// TIA Portal V17 export
// export: Created 2023-07-20T16:54:09.9633399Z, ExportSetting WithDefaults, DisplayName Totally Integrated Automation Portal, DisplayVersion V17, DisplayName TIA Portal Openness, DisplayVersion V17, DisplayName TIA Portal Version Control Interface, DisplayVersion V17, DisplayName STEP 7 Professional, DisplayVersion V17, DisplayName STEP 7 Safety, DisplayVersion V17, DisplayName WinCC Professional, DisplayVersion V17
FUNCTION_BLOCK "Modbus RTU RW sequencer"   // FB1, LAD
{ S7_Optimized_Access := 'TRUE' }
VERSION : 0.1
// stored: AutoNumber false, IsIECCheckEnabled false, IsRetainMemResEnabled false, MemoryReserve 100, SetENOAutomatically false, UDAEnableTagReadback false
   VAR
      "Operation data number" { S7_SetPoint := 'True'} : "Deconcatenate UDInt into two UInt";
      "Operation type" { S7_SetPoint := 'True'} : "Deconcatenate UDInt into two UInt";
      Position { S7_SetPoint := 'True'} : "Deconcatenate UDInt into two UInt";
      Speed { S7_SetPoint := 'True'} : "Deconcatenate UDInt into two UInt";
      "Starting changing rate" { S7_SetPoint := 'True'} : "Deconcatenate UDInt into two UInt";
      "Stopping deceleration" { S7_SetPoint := 'True'} : "Deconcatenate UDInt into two UInt";
      "Operating current" { S7_SetPoint := 'True'} : "Deconcatenate UDInt into two UInt";
      "Operation trigger" { S7_SetPoint := 'True'} : "Deconcatenate UDInt into two UInt";
      "Forwarding destination" { S7_SetPoint := 'True'} : "Deconcatenate UDInt into two UInt";
      "Alarm reset" { S7_SetPoint := 'True'} : "Deconcatenate UDInt into two UInt";
      "Clear alarm history" { S7_SetPoint := 'True'} : "Deconcatenate UDInt into two UInt";
      "Clear comm history" { S7_SetPoint := 'True'} : "Deconcatenate UDInt into two UInt";
      "Clear monitor alarm history" { S7_SetPoint := 'True'} : "Deconcatenate UDInt into two UInt";
      "Clear comm history_1" { S7_SetPoint := 'True'} : "Deconcatenate UDInt into two UInt";
      "Monitor present alarm" { S7_SetPoint := 'True'} : "Concatenate two UInt into one UDInt";
      "Monitor alarm history 1" { S7_SetPoint := 'True'} : "Concatenate two UInt into one UDInt";
      "Monitor alarm history 2" { S7_SetPoint := 'True'} : "Concatenate two UInt into one UDInt";
      "Monitor alarm history 3" { S7_SetPoint := 'True'} : "Concatenate two UInt into one UDInt";
      "Monitor alarm history 4" { S7_SetPoint := 'True'} : "Concatenate two UInt into one UDInt";
      "Monitor alarm history 5" { S7_SetPoint := 'True'} : "Concatenate two UInt into one UDInt";
      "Monitor present communication error" { S7_SetPoint := 'True'} : "Concatenate two UInt into one UDInt";
      "Monitor communication error history 1" { S7_SetPoint := 'True'} : "Concatenate two UInt into one UDInt";
      "Monitor communication error history 2" { S7_SetPoint := 'True'} : "Concatenate two UInt into one UDInt";
      "Monitor communication error history 3" { S7_SetPoint := 'True'} : "Concatenate two UInt into one UDInt";
      "Monitor communication error history 4" { S7_SetPoint := 'True'} : "Concatenate two UInt into one UDInt";
      "Monitor communication error history 5" { S7_SetPoint := 'True'} : "Concatenate two UInt into one UDInt";
      "Monitor feedback position" { S7_SetPoint := 'True'} : "Concatenate two UInt into one UDInt";
      "Monitor feedback speed r/min" { S7_SetPoint := 'True'} : "Concatenate two UInt into one UDInt";
      "Monitor feedback speed Hz" { S7_SetPoint := 'True'} : "Concatenate two UInt into one UDInt";
      "Monitor direct I/O" { S7_SetPoint := 'True'} : "Concatenate two UInt into one UDInt";
      "Monitor torque" { S7_SetPoint := 'True'} : "Concatenate two UInt into one UDInt";
      "Monitor cumulative load" { S7_SetPoint := 'True'} : "Concatenate two UInt into one UDInt";
      "Monitor driver temperature" { S7_SetPoint := 'True'} : "Concatenate two UInt into one UDInt";
      "Monitor motor temperature" { S7_SetPoint := 'True'} : "Concatenate two UInt into one UDInt";
      "Monitor inverter voltage" { S7_SetPoint := 'True'} : "Concatenate two UInt into one UDInt";
      "Monitor power supply voltage" { S7_SetPoint := 'True'} : "Concatenate two UInt into one UDInt";
      "Monitor DIP SW" { S7_SetPoint := 'True'} : "Concatenate two UInt into one UDInt";
      "Monitor ROT SW0" { S7_SetPoint := 'True'} : "Concatenate two UInt into one UDInt";
      "Monitor ROT SW1" { S7_SetPoint := 'True'} : "Concatenate two UInt into one UDInt";
   END_VAR
   VAR_TEMP   // added for the SCL form of the ladder/FBD networks
      _w1 : Bool;
   END_VAR
BEGIN

REGION Network 1: Deconcatenate data for writing it into modbus holding registers
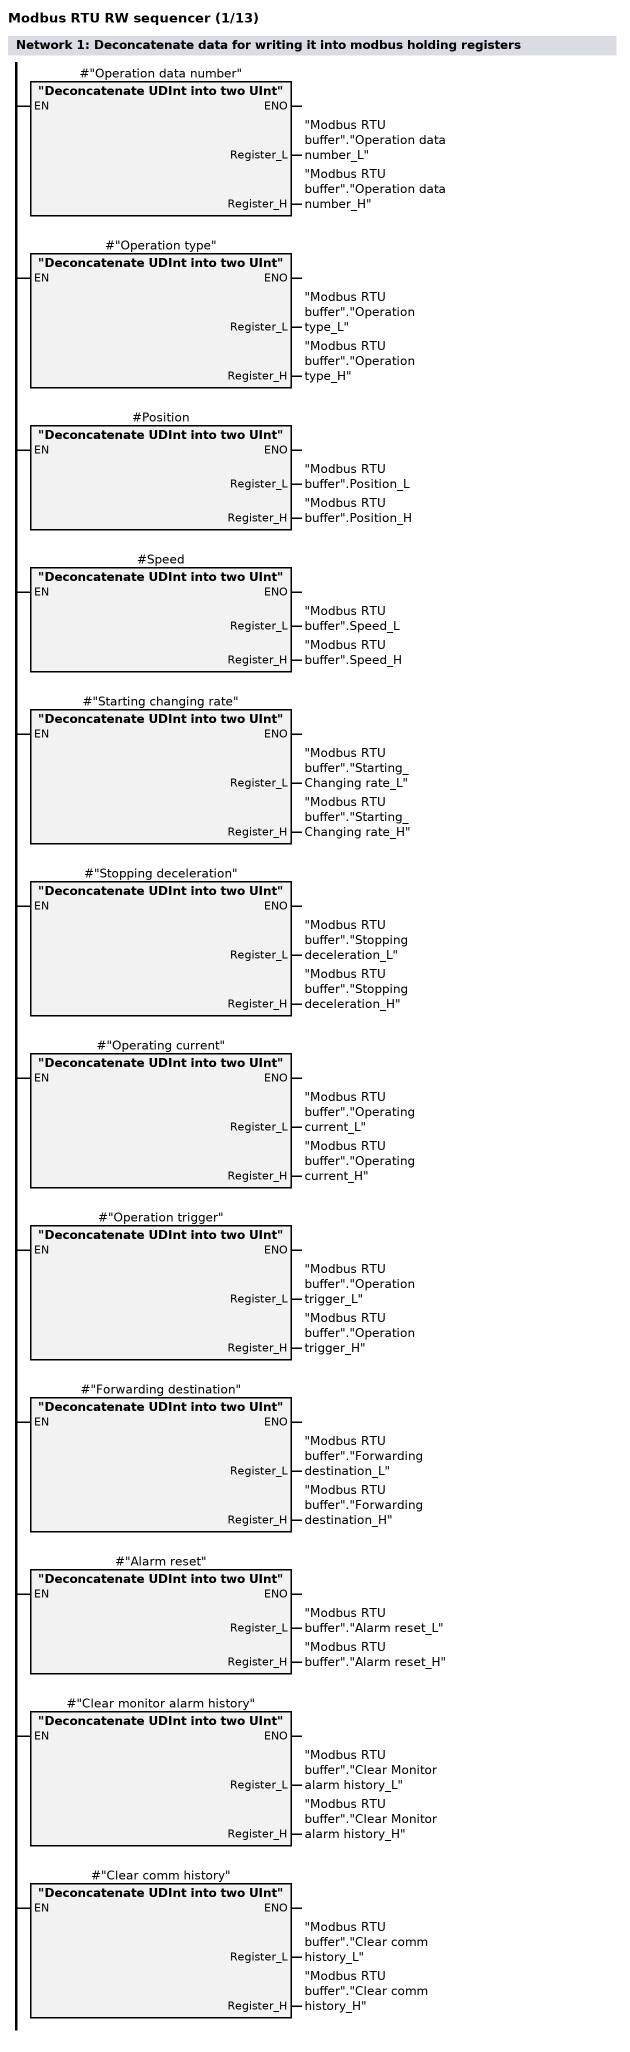
   RUNG wire#powerrail
      #"Operation data number"(Register_L => "Modbus RTU buffer"."Operation data number_L", Register_H => "Modbus RTU buffer"."Operation data number_H")
   END_RUNG
   RUNG wire#powerrail
      #"Operation type"(Register_L => "Modbus RTU buffer"."Operation type_L", Register_H => "Modbus RTU buffer"."Operation type_H")
   END_RUNG
   RUNG wire#powerrail
      #Position(Register_L => "Modbus RTU buffer".Position_L, Register_H => "Modbus RTU buffer".Position_H)
   END_RUNG
   RUNG wire#powerrail
      #Speed(Register_L => "Modbus RTU buffer".Speed_L, Register_H => "Modbus RTU buffer".Speed_H)
   END_RUNG
   RUNG wire#powerrail
      #"Starting changing rate"(Register_L => "Modbus RTU buffer"."Starting_Changing rate_L", Register_H => "Modbus RTU buffer"."Starting_Changing rate_H")
   END_RUNG
   RUNG wire#powerrail
      #"Stopping deceleration"(Register_L => "Modbus RTU buffer"."Stopping deceleration_L", Register_H => "Modbus RTU buffer"."Stopping deceleration_H")
   END_RUNG
   RUNG wire#powerrail
      #"Operating current"(Register_L => "Modbus RTU buffer"."Operating current_L", Register_H => "Modbus RTU buffer"."Operating current_H")
   END_RUNG
   RUNG wire#powerrail
      #"Operation trigger"(Register_L => "Modbus RTU buffer"."Operation trigger_L", Register_H => "Modbus RTU buffer"."Operation trigger_H")
   END_RUNG
   RUNG wire#powerrail
      #"Forwarding destination"(Register_L => "Modbus RTU buffer"."Forwarding destination_L", Register_H => "Modbus RTU buffer"."Forwarding destination_H")
   END_RUNG
   RUNG wire#powerrail
      #"Alarm reset"(Register_L => "Modbus RTU buffer"."Alarm reset_L", Register_H => "Modbus RTU buffer"."Alarm reset_H")
   END_RUNG
   RUNG wire#powerrail
      #"Clear monitor alarm history"(Register_L => "Modbus RTU buffer"."Clear Monitor alarm history_L", Register_H => "Modbus RTU buffer"."Clear Monitor alarm history_H")
   END_RUNG
   RUNG wire#powerrail
      #"Clear comm history"(Register_L => "Modbus RTU buffer"."Clear comm history_L", Register_H => "Modbus RTU buffer"."Clear comm history_H")
   END_RUNG
   // the same network as SCL:
   #"Operation data number"(Register_L => "Modbus RTU buffer"."Operation data number_L",   // "Deconcatenate UDInt into two UInt"
                           Register_H => "Modbus RTU buffer"."Operation data number_H");
   #"Operation type"(Register_L => "Modbus RTU buffer"."Operation type_L",   // "Deconcatenate UDInt into two UInt"
                     Register_H => "Modbus RTU buffer"."Operation type_H");
   #Position(Register_L => "Modbus RTU buffer".Position_L, Register_H => "Modbus RTU buffer".Position_H);   // "Deconcatenate UDInt into two UInt"
   #Speed(Register_L => "Modbus RTU buffer".Speed_L, Register_H => "Modbus RTU buffer".Speed_H);   // "Deconcatenate UDInt into two UInt"
   #"Starting changing rate"(Register_L => "Modbus RTU buffer"."Starting_Changing rate_L",   // "Deconcatenate UDInt into two UInt"
                           Register_H => "Modbus RTU buffer"."Starting_Changing rate_H");
   #"Stopping deceleration"(Register_L => "Modbus RTU buffer"."Stopping deceleration_L",   // "Deconcatenate UDInt into two UInt"
                           Register_H => "Modbus RTU buffer"."Stopping deceleration_H");
   #"Operating current"(Register_L => "Modbus RTU buffer"."Operating current_L",   // "Deconcatenate UDInt into two UInt"
                        Register_H => "Modbus RTU buffer"."Operating current_H");
   #"Operation trigger"(Register_L => "Modbus RTU buffer"."Operation trigger_L",   // "Deconcatenate UDInt into two UInt"
                        Register_H => "Modbus RTU buffer"."Operation trigger_H");
   #"Forwarding destination"(Register_L => "Modbus RTU buffer"."Forwarding destination_L",   // "Deconcatenate UDInt into two UInt"
                           Register_H => "Modbus RTU buffer"."Forwarding destination_H");
   #"Alarm reset"(Register_L => "Modbus RTU buffer"."Alarm reset_L",   // "Deconcatenate UDInt into two UInt"
                  Register_H => "Modbus RTU buffer"."Alarm reset_H");
   #"Clear monitor alarm history"(Register_L => "Modbus RTU buffer"."Clear Monitor alarm history_L",   // "Deconcatenate UDInt into two UInt"
                           Register_H => "Modbus RTU buffer"."Clear Monitor alarm history_H");
   #"Clear comm history"(Register_L => "Modbus RTU buffer"."Clear comm history_L",   // "Deconcatenate UDInt into two UInt"
                         Register_H => "Modbus RTU buffer"."Clear comm history_H");
END_REGION

REGION Network 2: Data writing/reading step 0: Write data from address 88 to address 105
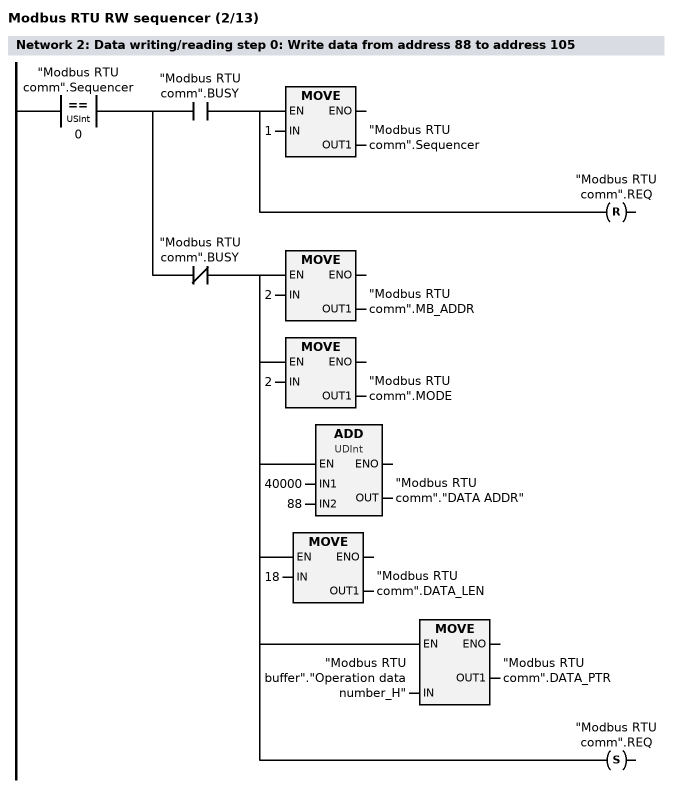
   RUNG wire#powerrail
      { S7_Templates := "SrcType := USInt" } EQ_Contact(in1 := "Modbus RTU comm".Sequencer, in2 := 0)
      wire#w1
      Contact( "Modbus RTU comm".BUSY )
      wire#w2
      Move(in := 1, out1 => "Modbus RTU comm".Sequencer)
   END_RUNG
   RUNG wire#w2
      R_Coil( "Modbus RTU comm".REQ )
   END_RUNG
   RUNG wire#w1
      I_Contact( "Modbus RTU comm".BUSY )
      wire#w3
      Move(in := 2, out1 => "Modbus RTU comm".MB_ADDR)
   END_RUNG
   RUNG wire#w3
      Move(in := 2, out1 => "Modbus RTU comm".MODE)
   END_RUNG
   RUNG wire#w3
      { S7_Templates := "SrcType := UDInt" } Add(in1 := 40000, in2 := 88, out => "Modbus RTU comm"."DATA ADDR")
   END_RUNG
   RUNG wire#w3
      Move(in := 18, out1 => "Modbus RTU comm".DATA_LEN)
   END_RUNG
   RUNG wire#w3
      Move(in := "Modbus RTU buffer"."Operation data number_H", out1 => "Modbus RTU comm".DATA_PTR)
   END_RUNG
   RUNG wire#w3
      S_Coil( "Modbus RTU comm".REQ )
   END_RUNG
   // the same network as SCL:
   #_w1 := "Modbus RTU comm".Sequencer = 0;
   IF #_w1 AND "Modbus RTU comm".BUSY THEN
       "Modbus RTU comm".Sequencer := 1;
       "Modbus RTU comm".REQ := FALSE;
   END_IF;
   IF #_w1 AND NOT "Modbus RTU comm".BUSY THEN
       "Modbus RTU comm".MB_ADDR := 2;
       "Modbus RTU comm".MODE := 2;
       "Modbus RTU comm"."DATA ADDR" := 40000 + 88;
       "Modbus RTU comm".DATA_LEN := 18;
       "Modbus RTU comm".DATA_PTR := "Modbus RTU buffer"."Operation data number_H";
       "Modbus RTU comm".REQ := TRUE;
   END_IF;
END_REGION

REGION Network 3: Data writing/reading step 1: Write data from address 384 to address 385
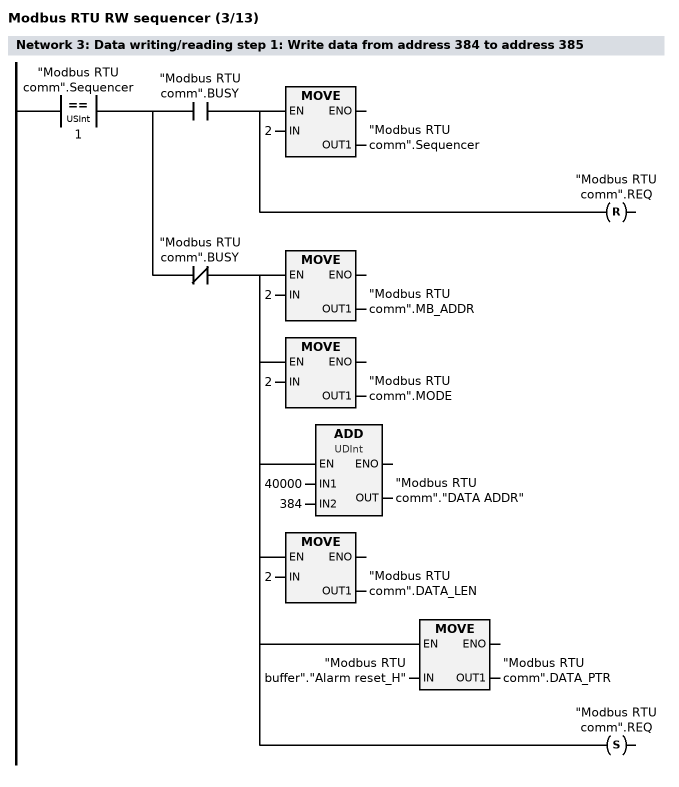
   RUNG wire#powerrail
      { S7_Templates := "SrcType := USInt" } EQ_Contact(in1 := "Modbus RTU comm".Sequencer, in2 := 1)
      wire#w1
      Contact( "Modbus RTU comm".BUSY )
      wire#w2
      Move(in := 2, out1 => "Modbus RTU comm".Sequencer)
   END_RUNG
   RUNG wire#w2
      R_Coil( "Modbus RTU comm".REQ )
   END_RUNG
   RUNG wire#w1
      I_Contact( "Modbus RTU comm".BUSY )
      wire#w3
      Move(in := 2, out1 => "Modbus RTU comm".MB_ADDR)
   END_RUNG
   RUNG wire#w3
      Move(in := 2, out1 => "Modbus RTU comm".MODE)
   END_RUNG
   RUNG wire#w3
      { S7_Templates := "SrcType := UDInt" } Add(in1 := 40000, in2 := 384, out => "Modbus RTU comm"."DATA ADDR")
   END_RUNG
   RUNG wire#w3
      Move(in := 2, out1 => "Modbus RTU comm".DATA_LEN)
   END_RUNG
   RUNG wire#w3
      Move(in := "Modbus RTU buffer"."Alarm reset_H", out1 => "Modbus RTU comm".DATA_PTR)
   END_RUNG
   RUNG wire#w3
      S_Coil( "Modbus RTU comm".REQ )
   END_RUNG
   // the same network as SCL:
   #_w1 := "Modbus RTU comm".Sequencer = 1;
   IF #_w1 AND "Modbus RTU comm".BUSY THEN
       "Modbus RTU comm".Sequencer := 2;
       "Modbus RTU comm".REQ := FALSE;
   END_IF;
   IF #_w1 AND NOT "Modbus RTU comm".BUSY THEN
       "Modbus RTU comm".MB_ADDR := 2;
       "Modbus RTU comm".MODE := 2;
       "Modbus RTU comm"."DATA ADDR" := 40000 + 384;
       "Modbus RTU comm".DATA_LEN := 2;
       "Modbus RTU comm".DATA_PTR := "Modbus RTU buffer"."Alarm reset_H";
       "Modbus RTU comm".REQ := TRUE;
   END_IF;
END_REGION

REGION Network 4: Data writing/reading step 2: Write data from address 388 to address 389
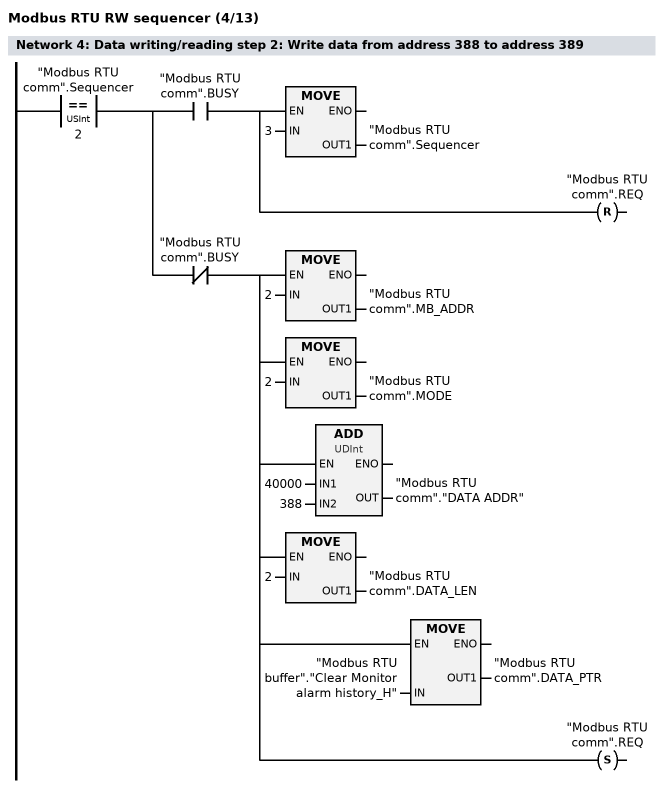
   RUNG wire#powerrail
      { S7_Templates := "SrcType := USInt" } EQ_Contact(in1 := "Modbus RTU comm".Sequencer, in2 := 2)
      wire#w1
      Contact( "Modbus RTU comm".BUSY )
      wire#w2
      Move(in := 3, out1 => "Modbus RTU comm".Sequencer)
   END_RUNG
   RUNG wire#w2
      R_Coil( "Modbus RTU comm".REQ )
   END_RUNG
   RUNG wire#w1
      I_Contact( "Modbus RTU comm".BUSY )
      wire#w3
      Move(in := 2, out1 => "Modbus RTU comm".MB_ADDR)
   END_RUNG
   RUNG wire#w3
      Move(in := 2, out1 => "Modbus RTU comm".MODE)
   END_RUNG
   RUNG wire#w3
      { S7_Templates := "SrcType := UDInt" } Add(in1 := 40000, in2 := 388, out => "Modbus RTU comm"."DATA ADDR")
   END_RUNG
   RUNG wire#w3
      Move(in := 2, out1 => "Modbus RTU comm".DATA_LEN)
   END_RUNG
   RUNG wire#w3
      Move(in := "Modbus RTU buffer"."Clear Monitor alarm history_H", out1 => "Modbus RTU comm".DATA_PTR)
   END_RUNG
   RUNG wire#w3
      S_Coil( "Modbus RTU comm".REQ )
   END_RUNG
   // the same network as SCL:
   #_w1 := "Modbus RTU comm".Sequencer = 2;
   IF #_w1 AND "Modbus RTU comm".BUSY THEN
       "Modbus RTU comm".Sequencer := 3;
       "Modbus RTU comm".REQ := FALSE;
   END_IF;
   IF #_w1 AND NOT "Modbus RTU comm".BUSY THEN
       "Modbus RTU comm".MB_ADDR := 2;
       "Modbus RTU comm".MODE := 2;
       "Modbus RTU comm"."DATA ADDR" := 40000 + 388;
       "Modbus RTU comm".DATA_LEN := 2;
       "Modbus RTU comm".DATA_PTR := "Modbus RTU buffer"."Clear Monitor alarm history_H";
       "Modbus RTU comm".REQ := TRUE;
   END_IF;
END_REGION

REGION Network 5: Data writing/reading step 3: Write data from address 392 to address 393
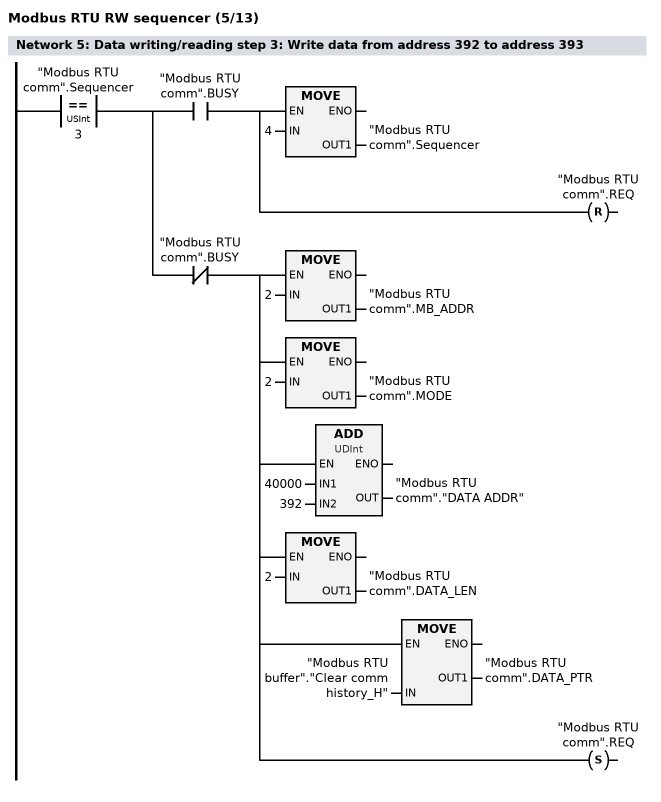
   RUNG wire#powerrail
      { S7_Templates := "SrcType := USInt" } EQ_Contact(in1 := "Modbus RTU comm".Sequencer, in2 := 3)
      wire#w1
      Contact( "Modbus RTU comm".BUSY )
      wire#w2
      Move(in := 4, out1 => "Modbus RTU comm".Sequencer)
   END_RUNG
   RUNG wire#w2
      R_Coil( "Modbus RTU comm".REQ )
   END_RUNG
   RUNG wire#w1
      I_Contact( "Modbus RTU comm".BUSY )
      wire#w3
      Move(in := 2, out1 => "Modbus RTU comm".MB_ADDR)
   END_RUNG
   RUNG wire#w3
      Move(in := 2, out1 => "Modbus RTU comm".MODE)
   END_RUNG
   RUNG wire#w3
      { S7_Templates := "SrcType := UDInt" } Add(in1 := 40000, in2 := 392, out => "Modbus RTU comm"."DATA ADDR")
   END_RUNG
   RUNG wire#w3
      Move(in := 2, out1 => "Modbus RTU comm".DATA_LEN)
   END_RUNG
   RUNG wire#w3
      Move(in := "Modbus RTU buffer"."Clear comm history_H", out1 => "Modbus RTU comm".DATA_PTR)
   END_RUNG
   RUNG wire#w3
      S_Coil( "Modbus RTU comm".REQ )
   END_RUNG
   // the same network as SCL:
   #_w1 := "Modbus RTU comm".Sequencer = 3;
   IF #_w1 AND "Modbus RTU comm".BUSY THEN
       "Modbus RTU comm".Sequencer := 4;
       "Modbus RTU comm".REQ := FALSE;
   END_IF;
   IF #_w1 AND NOT "Modbus RTU comm".BUSY THEN
       "Modbus RTU comm".MB_ADDR := 2;
       "Modbus RTU comm".MODE := 2;
       "Modbus RTU comm"."DATA ADDR" := 40000 + 392;
       "Modbus RTU comm".DATA_LEN := 2;
       "Modbus RTU comm".DATA_PTR := "Modbus RTU buffer"."Clear comm history_H";
       "Modbus RTU comm".REQ := TRUE;
   END_IF;
END_REGION

REGION Network 6: Data writing/reading step 4: Read data from address 128 to address 139
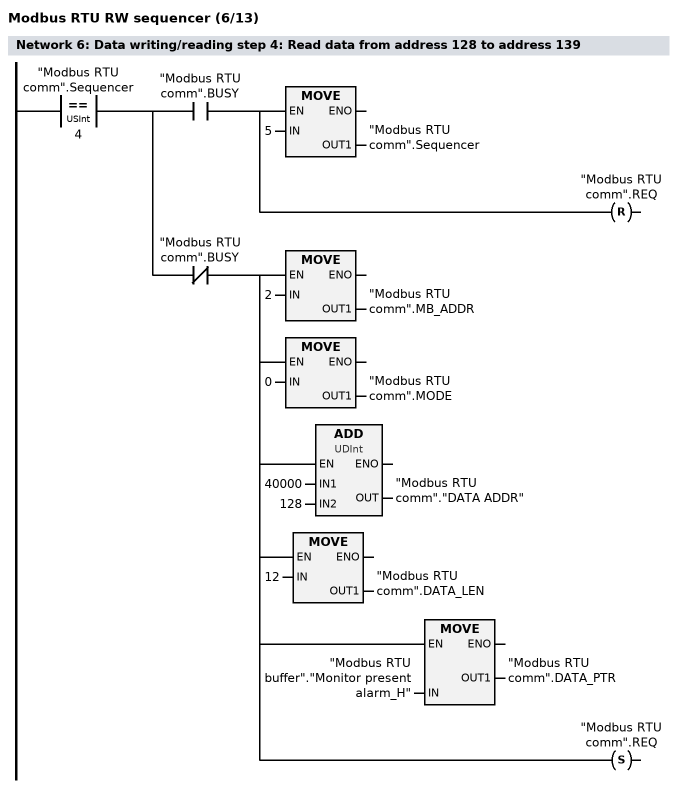
   RUNG wire#powerrail
      { S7_Templates := "SrcType := USInt" } EQ_Contact(in1 := "Modbus RTU comm".Sequencer, in2 := 4)
      wire#w1
      Contact( "Modbus RTU comm".BUSY )
      wire#w2
      Move(in := 5, out1 => "Modbus RTU comm".Sequencer)
   END_RUNG
   RUNG wire#w2
      R_Coil( "Modbus RTU comm".REQ )
   END_RUNG
   RUNG wire#w1
      I_Contact( "Modbus RTU comm".BUSY )
      wire#w3
      Move(in := 2, out1 => "Modbus RTU comm".MB_ADDR)
   END_RUNG
   RUNG wire#w3
      Move(in := 0, out1 => "Modbus RTU comm".MODE)
   END_RUNG
   RUNG wire#w3
      { S7_Templates := "SrcType := UDInt" } Add(in1 := 40000, in2 := 128, out => "Modbus RTU comm"."DATA ADDR")
   END_RUNG
   RUNG wire#w3
      Move(in := 12, out1 => "Modbus RTU comm".DATA_LEN)
   END_RUNG
   RUNG wire#w3
      Move(in := "Modbus RTU buffer"."Monitor present alarm_H", out1 => "Modbus RTU comm".DATA_PTR)
   END_RUNG
   RUNG wire#w3
      S_Coil( "Modbus RTU comm".REQ )
   END_RUNG
   // the same network as SCL:
   #_w1 := "Modbus RTU comm".Sequencer = 4;
   IF #_w1 AND "Modbus RTU comm".BUSY THEN
       "Modbus RTU comm".Sequencer := 5;
       "Modbus RTU comm".REQ := FALSE;
   END_IF;
   IF #_w1 AND NOT "Modbus RTU comm".BUSY THEN
       "Modbus RTU comm".MB_ADDR := 2;
       "Modbus RTU comm".MODE := 0;
       "Modbus RTU comm"."DATA ADDR" := 40000 + 128;
       "Modbus RTU comm".DATA_LEN := 12;
       "Modbus RTU comm".DATA_PTR := "Modbus RTU buffer"."Monitor present alarm_H";
       "Modbus RTU comm".REQ := TRUE;
   END_IF;
END_REGION

REGION Network 7: Data writing/reading step 5: Read data from address 172 to address 183
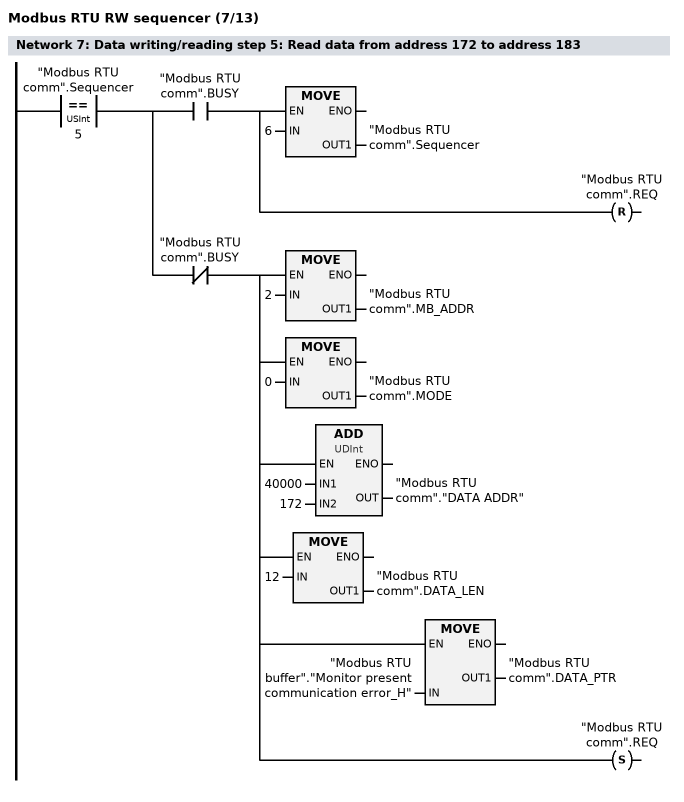
   RUNG wire#powerrail
      { S7_Templates := "SrcType := USInt" } EQ_Contact(in1 := "Modbus RTU comm".Sequencer, in2 := 5)
      wire#w1
      Contact( "Modbus RTU comm".BUSY )
      wire#w2
      Move(in := 6, out1 => "Modbus RTU comm".Sequencer)
   END_RUNG
   RUNG wire#w2
      R_Coil( "Modbus RTU comm".REQ )
   END_RUNG
   RUNG wire#w1
      I_Contact( "Modbus RTU comm".BUSY )
      wire#w3
      Move(in := 2, out1 => "Modbus RTU comm".MB_ADDR)
   END_RUNG
   RUNG wire#w3
      Move(in := 0, out1 => "Modbus RTU comm".MODE)
   END_RUNG
   RUNG wire#w3
      { S7_Templates := "SrcType := UDInt" } Add(in1 := 40000, in2 := 172, out => "Modbus RTU comm"."DATA ADDR")
   END_RUNG
   RUNG wire#w3
      Move(in := 12, out1 => "Modbus RTU comm".DATA_LEN)
   END_RUNG
   RUNG wire#w3
      Move(in := "Modbus RTU buffer"."Monitor present communication error_H", out1 => "Modbus RTU comm".DATA_PTR)
   END_RUNG
   RUNG wire#w3
      S_Coil( "Modbus RTU comm".REQ )
   END_RUNG
   // the same network as SCL:
   #_w1 := "Modbus RTU comm".Sequencer = 5;
   IF #_w1 AND "Modbus RTU comm".BUSY THEN
       "Modbus RTU comm".Sequencer := 6;
       "Modbus RTU comm".REQ := FALSE;
   END_IF;
   IF #_w1 AND NOT "Modbus RTU comm".BUSY THEN
       "Modbus RTU comm".MB_ADDR := 2;
       "Modbus RTU comm".MODE := 0;
       "Modbus RTU comm"."DATA ADDR" := 40000 + 172;
       "Modbus RTU comm".DATA_LEN := 12;
       "Modbus RTU comm".DATA_PTR := "Modbus RTU buffer"."Monitor present communication error_H";
       "Modbus RTU comm".REQ := TRUE;
   END_IF;
END_REGION

REGION Network 8: Data writing/reading step 6: Read data from address 204 to address 209
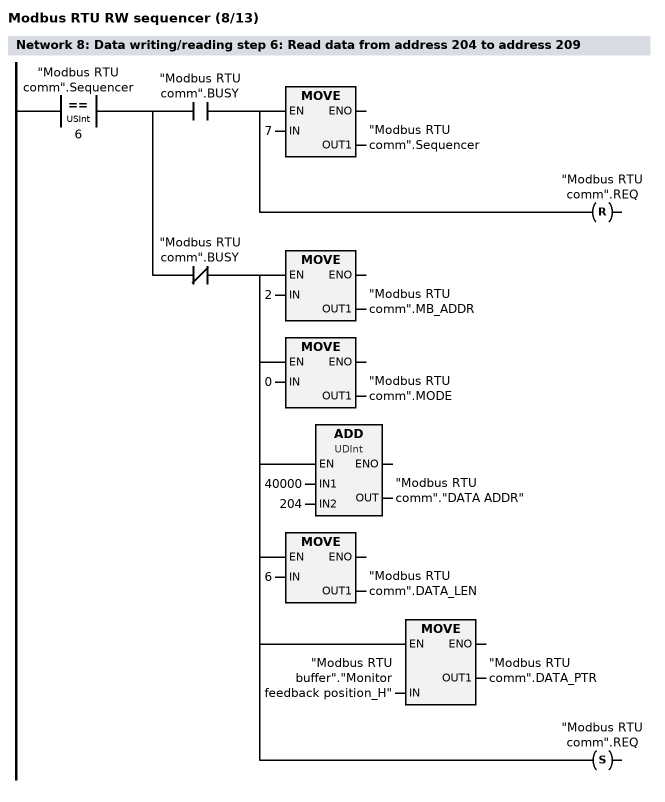
   RUNG wire#powerrail
      { S7_Templates := "SrcType := USInt" } EQ_Contact(in1 := "Modbus RTU comm".Sequencer, in2 := 6)
      wire#w1
      Contact( "Modbus RTU comm".BUSY )
      wire#w2
      Move(in := 7, out1 => "Modbus RTU comm".Sequencer)
   END_RUNG
   RUNG wire#w2
      R_Coil( "Modbus RTU comm".REQ )
   END_RUNG
   RUNG wire#w1
      I_Contact( "Modbus RTU comm".BUSY )
      wire#w3
      Move(in := 2, out1 => "Modbus RTU comm".MB_ADDR)
   END_RUNG
   RUNG wire#w3
      Move(in := 0, out1 => "Modbus RTU comm".MODE)
   END_RUNG
   RUNG wire#w3
      { S7_Templates := "SrcType := UDInt" } Add(in1 := 40000, in2 := 204, out => "Modbus RTU comm"."DATA ADDR")
   END_RUNG
   RUNG wire#w3
      Move(in := 6, out1 => "Modbus RTU comm".DATA_LEN)
   END_RUNG
   RUNG wire#w3
      Move(in := "Modbus RTU buffer"."Monitor feedback position_H", out1 => "Modbus RTU comm".DATA_PTR)
   END_RUNG
   RUNG wire#w3
      S_Coil( "Modbus RTU comm".REQ )
   END_RUNG
   // the same network as SCL:
   #_w1 := "Modbus RTU comm".Sequencer = 6;
   IF #_w1 AND "Modbus RTU comm".BUSY THEN
       "Modbus RTU comm".Sequencer := 7;
       "Modbus RTU comm".REQ := FALSE;
   END_IF;
   IF #_w1 AND NOT "Modbus RTU comm".BUSY THEN
       "Modbus RTU comm".MB_ADDR := 2;
       "Modbus RTU comm".MODE := 0;
       "Modbus RTU comm"."DATA ADDR" := 40000 + 204;
       "Modbus RTU comm".DATA_LEN := 6;
       "Modbus RTU comm".DATA_PTR := "Modbus RTU buffer"."Monitor feedback position_H";
       "Modbus RTU comm".REQ := TRUE;
   END_IF;
END_REGION

REGION Network 9: Data writing/reading step 7: Read data from address 212 to address 215
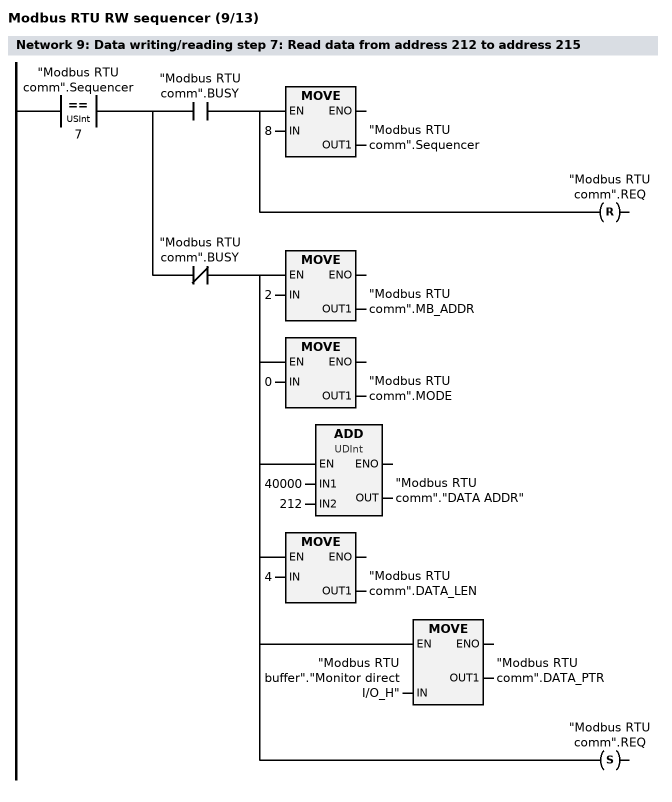
   RUNG wire#powerrail
      { S7_Templates := "SrcType := USInt" } EQ_Contact(in1 := "Modbus RTU comm".Sequencer, in2 := 7)
      wire#w1
      Contact( "Modbus RTU comm".BUSY )
      wire#w2
      Move(in := 8, out1 => "Modbus RTU comm".Sequencer)
   END_RUNG
   RUNG wire#w2
      R_Coil( "Modbus RTU comm".REQ )
   END_RUNG
   RUNG wire#w1
      I_Contact( "Modbus RTU comm".BUSY )
      wire#w3
      Move(in := 2, out1 => "Modbus RTU comm".MB_ADDR)
   END_RUNG
   RUNG wire#w3
      Move(in := 0, out1 => "Modbus RTU comm".MODE)
   END_RUNG
   RUNG wire#w3
      { S7_Templates := "SrcType := UDInt" } Add(in1 := 40000, in2 := 212, out => "Modbus RTU comm"."DATA ADDR")
   END_RUNG
   RUNG wire#w3
      Move(in := 4, out1 => "Modbus RTU comm".DATA_LEN)
   END_RUNG
   RUNG wire#w3
      Move(in := "Modbus RTU buffer"."Monitor direct I/O_H", out1 => "Modbus RTU comm".DATA_PTR)
   END_RUNG
   RUNG wire#w3
      S_Coil( "Modbus RTU comm".REQ )
   END_RUNG
   // the same network as SCL:
   #_w1 := "Modbus RTU comm".Sequencer = 7;
   IF #_w1 AND "Modbus RTU comm".BUSY THEN
       "Modbus RTU comm".Sequencer := 8;
       "Modbus RTU comm".REQ := FALSE;
   END_IF;
   IF #_w1 AND NOT "Modbus RTU comm".BUSY THEN
       "Modbus RTU comm".MB_ADDR := 2;
       "Modbus RTU comm".MODE := 0;
       "Modbus RTU comm"."DATA ADDR" := 40000 + 212;
       "Modbus RTU comm".DATA_LEN := 4;
       "Modbus RTU comm".DATA_PTR := "Modbus RTU buffer"."Monitor direct I/O_H";
       "Modbus RTU comm".REQ := TRUE;
   END_IF;
END_REGION

REGION Network 10: Data writing/reading step 8: Read data from address 218 to address 219
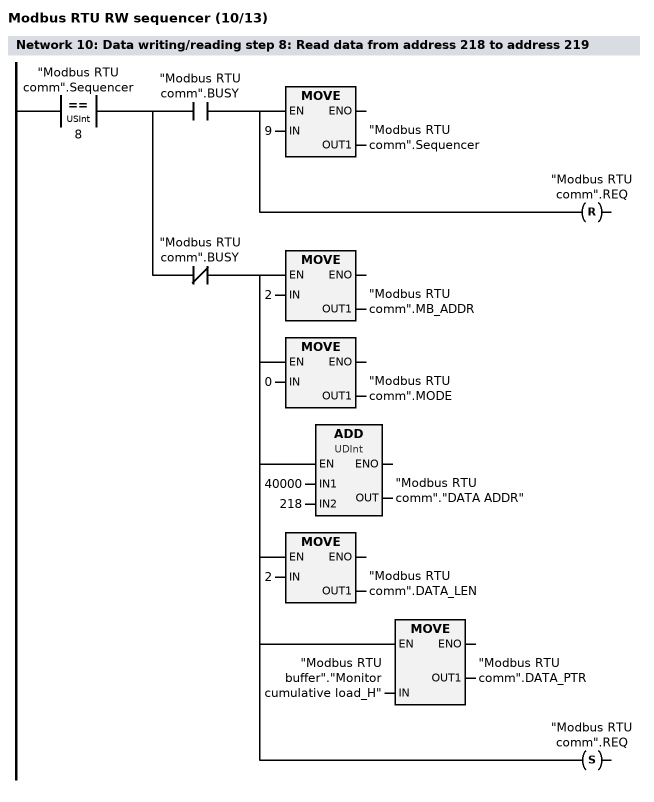
   RUNG wire#powerrail
      { S7_Templates := "SrcType := USInt" } EQ_Contact(in1 := "Modbus RTU comm".Sequencer, in2 := 8)
      wire#w1
      Contact( "Modbus RTU comm".BUSY )
      wire#w2
      Move(in := 9, out1 => "Modbus RTU comm".Sequencer)
   END_RUNG
   RUNG wire#w2
      R_Coil( "Modbus RTU comm".REQ )
   END_RUNG
   RUNG wire#w1
      I_Contact( "Modbus RTU comm".BUSY )
      wire#w3
      Move(in := 2, out1 => "Modbus RTU comm".MB_ADDR)
   END_RUNG
   RUNG wire#w3
      Move(in := 0, out1 => "Modbus RTU comm".MODE)
   END_RUNG
   RUNG wire#w3
      { S7_Templates := "SrcType := UDInt" } Add(in1 := 40000, in2 := 218, out => "Modbus RTU comm"."DATA ADDR")
   END_RUNG
   RUNG wire#w3
      Move(in := 2, out1 => "Modbus RTU comm".DATA_LEN)
   END_RUNG
   RUNG wire#w3
      Move(in := "Modbus RTU buffer"."Monitor cumulative load_H", out1 => "Modbus RTU comm".DATA_PTR)
   END_RUNG
   RUNG wire#w3
      S_Coil( "Modbus RTU comm".REQ )
   END_RUNG
   // the same network as SCL:
   #_w1 := "Modbus RTU comm".Sequencer = 8;
   IF #_w1 AND "Modbus RTU comm".BUSY THEN
       "Modbus RTU comm".Sequencer := 9;
       "Modbus RTU comm".REQ := FALSE;
   END_IF;
   IF #_w1 AND NOT "Modbus RTU comm".BUSY THEN
       "Modbus RTU comm".MB_ADDR := 2;
       "Modbus RTU comm".MODE := 0;
       "Modbus RTU comm"."DATA ADDR" := 40000 + 218;
       "Modbus RTU comm".DATA_LEN := 2;
       "Modbus RTU comm".DATA_PTR := "Modbus RTU buffer"."Monitor cumulative load_H";
       "Modbus RTU comm".REQ := TRUE;
   END_IF;
END_REGION

REGION Network 11: Data writing/reading step 9: Read data from address 248 to address 251
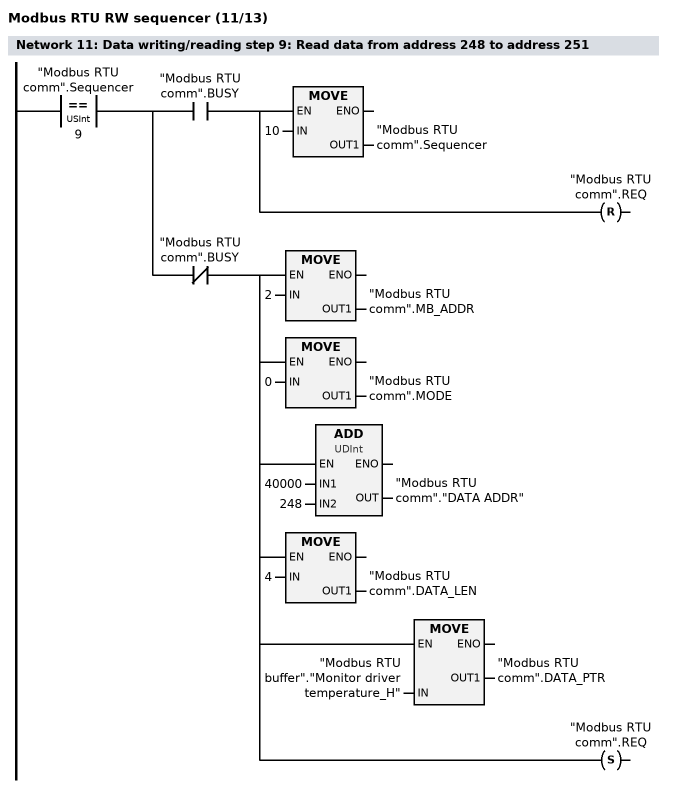
   RUNG wire#powerrail
      { S7_Templates := "SrcType := USInt" } EQ_Contact(in1 := "Modbus RTU comm".Sequencer, in2 := 9)
      wire#w1
      Contact( "Modbus RTU comm".BUSY )
      wire#w2
      Move(in := 10, out1 => "Modbus RTU comm".Sequencer)
   END_RUNG
   RUNG wire#w2
      R_Coil( "Modbus RTU comm".REQ )
   END_RUNG
   RUNG wire#w1
      I_Contact( "Modbus RTU comm".BUSY )
      wire#w3
      Move(in := 2, out1 => "Modbus RTU comm".MB_ADDR)
   END_RUNG
   RUNG wire#w3
      Move(in := 0, out1 => "Modbus RTU comm".MODE)
   END_RUNG
   RUNG wire#w3
      { S7_Templates := "SrcType := UDInt" } Add(in1 := 40000, in2 := 248, out => "Modbus RTU comm"."DATA ADDR")
   END_RUNG
   RUNG wire#w3
      Move(in := 4, out1 => "Modbus RTU comm".DATA_LEN)
   END_RUNG
   RUNG wire#w3
      Move(in := "Modbus RTU buffer"."Monitor driver temperature_H", out1 => "Modbus RTU comm".DATA_PTR)
   END_RUNG
   RUNG wire#w3
      S_Coil( "Modbus RTU comm".REQ )
   END_RUNG
   // the same network as SCL:
   #_w1 := "Modbus RTU comm".Sequencer = 9;
   IF #_w1 AND "Modbus RTU comm".BUSY THEN
       "Modbus RTU comm".Sequencer := 10;
       "Modbus RTU comm".REQ := FALSE;
   END_IF;
   IF #_w1 AND NOT "Modbus RTU comm".BUSY THEN
       "Modbus RTU comm".MB_ADDR := 2;
       "Modbus RTU comm".MODE := 0;
       "Modbus RTU comm"."DATA ADDR" := 40000 + 248;
       "Modbus RTU comm".DATA_LEN := 4;
       "Modbus RTU comm".DATA_PTR := "Modbus RTU buffer"."Monitor driver temperature_H";
       "Modbus RTU comm".REQ := TRUE;
   END_IF;
END_REGION

REGION Network 12: Data writing/reading step 10: Read data from address 326 to address 335
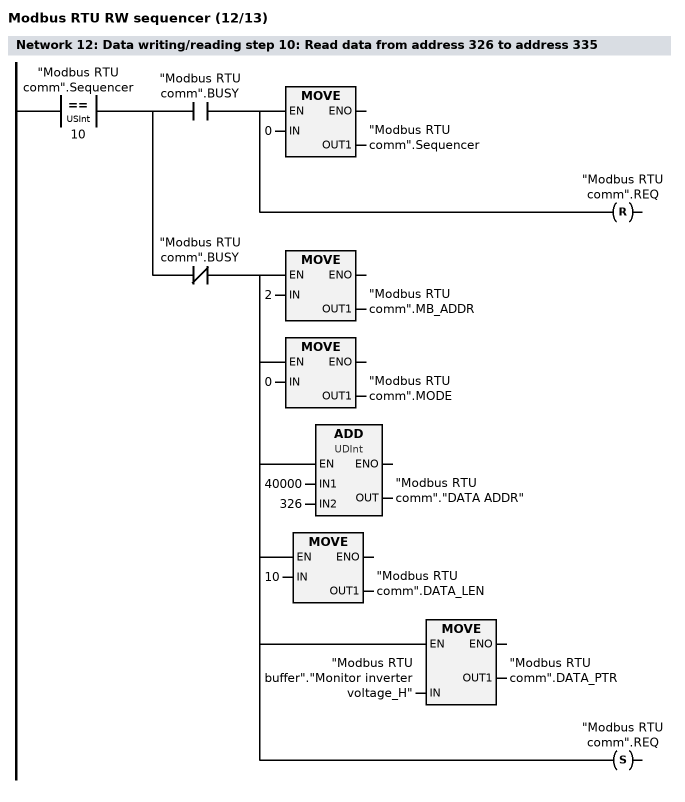
   RUNG wire#powerrail
      { S7_Templates := "SrcType := USInt" } EQ_Contact(in1 := "Modbus RTU comm".Sequencer, in2 := 10)
      wire#w1
      Contact( "Modbus RTU comm".BUSY )
      wire#w2
      Move(in := 0, out1 => "Modbus RTU comm".Sequencer)
   END_RUNG
   RUNG wire#w2
      R_Coil( "Modbus RTU comm".REQ )
   END_RUNG
   RUNG wire#w1
      I_Contact( "Modbus RTU comm".BUSY )
      wire#w3
      Move(in := 2, out1 => "Modbus RTU comm".MB_ADDR)
   END_RUNG
   RUNG wire#w3
      Move(in := 0, out1 => "Modbus RTU comm".MODE)
   END_RUNG
   RUNG wire#w3
      { S7_Templates := "SrcType := UDInt" } Add(in1 := 40000, in2 := 326, out => "Modbus RTU comm"."DATA ADDR")
   END_RUNG
   RUNG wire#w3
      Move(in := 10, out1 => "Modbus RTU comm".DATA_LEN)
   END_RUNG
   RUNG wire#w3
      Move(in := "Modbus RTU buffer"."Monitor inverter voltage_H", out1 => "Modbus RTU comm".DATA_PTR)
   END_RUNG
   RUNG wire#w3
      S_Coil( "Modbus RTU comm".REQ )
   END_RUNG
   // the same network as SCL:
   #_w1 := "Modbus RTU comm".Sequencer = 10;
   IF #_w1 AND "Modbus RTU comm".BUSY THEN
       "Modbus RTU comm".Sequencer := 0;
       "Modbus RTU comm".REQ := FALSE;
   END_IF;
   IF #_w1 AND NOT "Modbus RTU comm".BUSY THEN
       "Modbus RTU comm".MB_ADDR := 2;
       "Modbus RTU comm".MODE := 0;
       "Modbus RTU comm"."DATA ADDR" := 40000 + 326;
       "Modbus RTU comm".DATA_LEN := 10;
       "Modbus RTU comm".DATA_PTR := "Modbus RTU buffer"."Monitor inverter voltage_H";
       "Modbus RTU comm".REQ := TRUE;
   END_IF;
END_REGION

REGION Network 13: Concatenate data read from modbus holding registers into individual registers
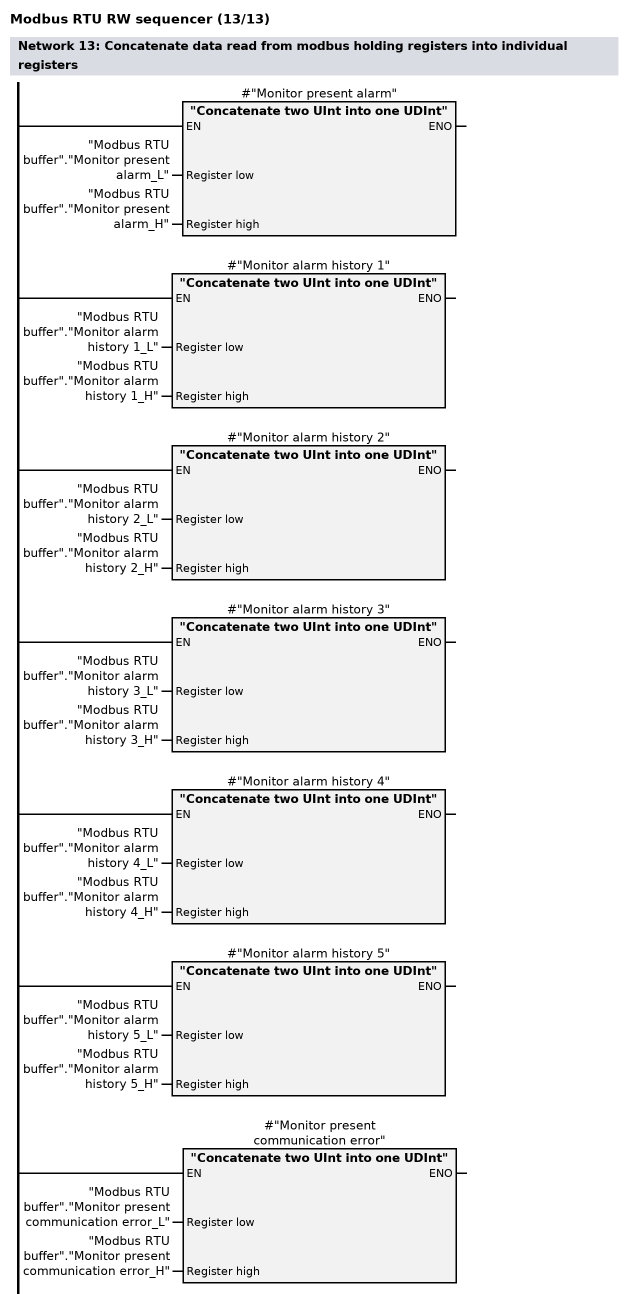
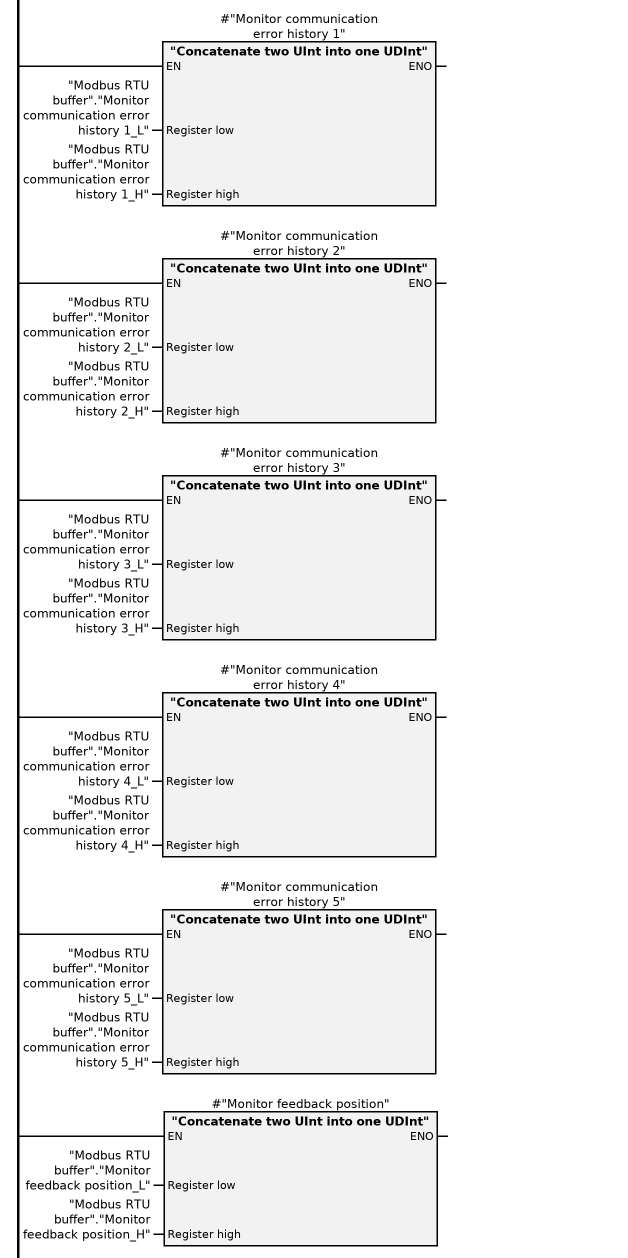
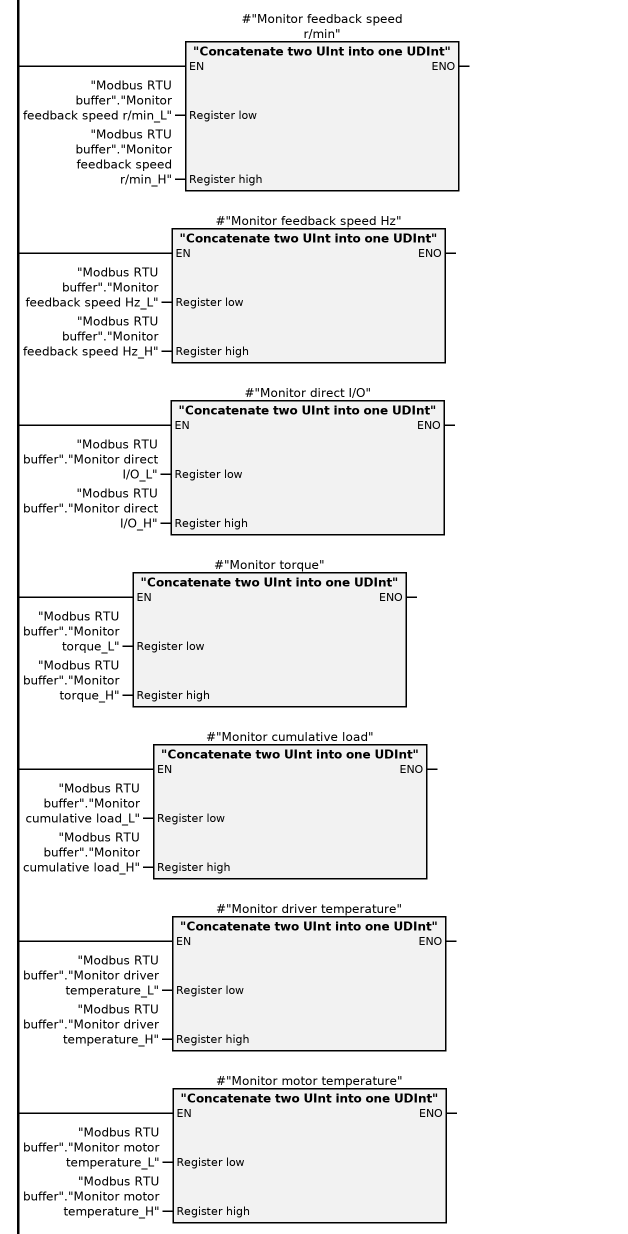
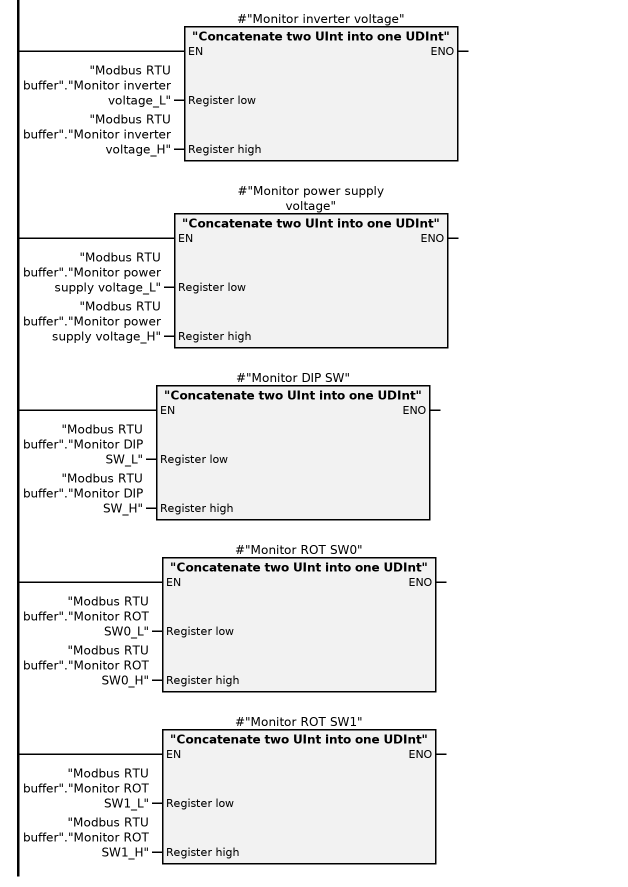
   RUNG wire#powerrail
      #"Monitor present alarm"("Register low" := "Modbus RTU buffer"."Monitor present alarm_L", "Register high" := "Modbus RTU buffer"."Monitor present alarm_H")
   END_RUNG
   RUNG wire#powerrail
      #"Monitor alarm history 1"("Register low" := "Modbus RTU buffer"."Monitor alarm history 1_L", "Register high" := "Modbus RTU buffer"."Monitor alarm history 1_H")
   END_RUNG
   RUNG wire#powerrail
      #"Monitor alarm history 2"("Register low" := "Modbus RTU buffer"."Monitor alarm history 2_L", "Register high" := "Modbus RTU buffer"."Monitor alarm history 2_H")
   END_RUNG
   RUNG wire#powerrail
      #"Monitor alarm history 3"("Register low" := "Modbus RTU buffer"."Monitor alarm history 3_L", "Register high" := "Modbus RTU buffer"."Monitor alarm history 3_H")
   END_RUNG
   RUNG wire#powerrail
      #"Monitor alarm history 4"("Register low" := "Modbus RTU buffer"."Monitor alarm history 4_L", "Register high" := "Modbus RTU buffer"."Monitor alarm history 4_H")
   END_RUNG
   RUNG wire#powerrail
      #"Monitor alarm history 5"("Register low" := "Modbus RTU buffer"."Monitor alarm history 5_L", "Register high" := "Modbus RTU buffer"."Monitor alarm history 5_H")
   END_RUNG
   RUNG wire#powerrail
      #"Monitor present communication error"("Register low" := "Modbus RTU buffer"."Monitor present communication error_L", "Register high" := "Modbus RTU buffer"."Monitor present communication error_H")
   END_RUNG
   RUNG wire#powerrail
      #"Monitor communication error history 1"("Register low" := "Modbus RTU buffer"."Monitor communication error history 1_L", "Register high" := "Modbus RTU buffer"."Monitor communication error history 1_H")
   END_RUNG
   RUNG wire#powerrail
      #"Monitor communication error history 2"("Register low" := "Modbus RTU buffer"."Monitor communication error history 2_L", "Register high" := "Modbus RTU buffer"."Monitor communication error history 2_H")
   END_RUNG
   RUNG wire#powerrail
      #"Monitor communication error history 3"("Register low" := "Modbus RTU buffer"."Monitor communication error history 3_L", "Register high" := "Modbus RTU buffer"."Monitor communication error history 3_H")
   END_RUNG
   RUNG wire#powerrail
      #"Monitor communication error history 4"("Register low" := "Modbus RTU buffer"."Monitor communication error history 4_L", "Register high" := "Modbus RTU buffer"."Monitor communication error history 4_H")
   END_RUNG
   RUNG wire#powerrail
      #"Monitor communication error history 5"("Register low" := "Modbus RTU buffer"."Monitor communication error history 5_L", "Register high" := "Modbus RTU buffer"."Monitor communication error history 5_H")
   END_RUNG
   RUNG wire#powerrail
      #"Monitor feedback position"("Register low" := "Modbus RTU buffer"."Monitor feedback position_L", "Register high" := "Modbus RTU buffer"."Monitor feedback position_H")
   END_RUNG
   RUNG wire#powerrail
      #"Monitor feedback speed r/min"("Register low" := "Modbus RTU buffer"."Monitor feedback speed r/min_L", "Register high" := "Modbus RTU buffer"."Monitor feedback speed r/min_H")
   END_RUNG
   RUNG wire#powerrail
      #"Monitor feedback speed Hz"("Register low" := "Modbus RTU buffer"."Monitor feedback speed Hz_L", "Register high" := "Modbus RTU buffer"."Monitor feedback speed Hz_H")
   END_RUNG
   RUNG wire#powerrail
      #"Monitor direct I/O"("Register low" := "Modbus RTU buffer"."Monitor direct I/O_L", "Register high" := "Modbus RTU buffer"."Monitor direct I/O_H")
   END_RUNG
   RUNG wire#powerrail
      #"Monitor torque"("Register low" := "Modbus RTU buffer"."Monitor torque_L", "Register high" := "Modbus RTU buffer"."Monitor torque_H")
   END_RUNG
   RUNG wire#powerrail
      #"Monitor cumulative load"("Register low" := "Modbus RTU buffer"."Monitor cumulative load_L", "Register high" := "Modbus RTU buffer"."Monitor cumulative load_H")
   END_RUNG
   RUNG wire#powerrail
      #"Monitor driver temperature"("Register low" := "Modbus RTU buffer"."Monitor driver temperature_L", "Register high" := "Modbus RTU buffer"."Monitor driver temperature_H")
   END_RUNG
   RUNG wire#powerrail
      #"Monitor motor temperature"("Register low" := "Modbus RTU buffer"."Monitor motor temperature_L", "Register high" := "Modbus RTU buffer"."Monitor motor temperature_H")
   END_RUNG
   RUNG wire#powerrail
      #"Monitor inverter voltage"("Register low" := "Modbus RTU buffer"."Monitor inverter voltage_L", "Register high" := "Modbus RTU buffer"."Monitor inverter voltage_H")
   END_RUNG
   RUNG wire#powerrail
      #"Monitor power supply voltage"("Register low" := "Modbus RTU buffer"."Monitor power supply voltage_L", "Register high" := "Modbus RTU buffer"."Monitor power supply voltage_H")
   END_RUNG
   RUNG wire#powerrail
      #"Monitor DIP SW"("Register low" := "Modbus RTU buffer"."Monitor DIP SW_L", "Register high" := "Modbus RTU buffer"."Monitor DIP SW_H")
   END_RUNG
   RUNG wire#powerrail
      #"Monitor ROT SW0"("Register low" := "Modbus RTU buffer"."Monitor ROT SW0_L", "Register high" := "Modbus RTU buffer"."Monitor ROT SW0_H")
   END_RUNG
   RUNG wire#powerrail
      #"Monitor ROT SW1"("Register low" := "Modbus RTU buffer"."Monitor ROT SW1_L", "Register high" := "Modbus RTU buffer"."Monitor ROT SW1_H")
   END_RUNG
   // the same network as SCL:
   #"Monitor present alarm"("Register low" := "Modbus RTU buffer"."Monitor present alarm_L",   // "Concatenate two UInt into one UDInt"
                           "Register high" := "Modbus RTU buffer"."Monitor present alarm_H");
   #"Monitor alarm history 1"("Register low" := "Modbus RTU buffer"."Monitor alarm history 1_L",   // "Concatenate two UInt into one UDInt"
                           "Register high" := "Modbus RTU buffer"."Monitor alarm history 1_H");
   #"Monitor alarm history 2"("Register low" := "Modbus RTU buffer"."Monitor alarm history 2_L",   // "Concatenate two UInt into one UDInt"
                           "Register high" := "Modbus RTU buffer"."Monitor alarm history 2_H");
   #"Monitor alarm history 3"("Register low" := "Modbus RTU buffer"."Monitor alarm history 3_L",   // "Concatenate two UInt into one UDInt"
                           "Register high" := "Modbus RTU buffer"."Monitor alarm history 3_H");
   #"Monitor alarm history 4"("Register low" := "Modbus RTU buffer"."Monitor alarm history 4_L",   // "Concatenate two UInt into one UDInt"
                           "Register high" := "Modbus RTU buffer"."Monitor alarm history 4_H");
   #"Monitor alarm history 5"("Register low" := "Modbus RTU buffer"."Monitor alarm history 5_L",   // "Concatenate two UInt into one UDInt"
                           "Register high" := "Modbus RTU buffer"."Monitor alarm history 5_H");
   #"Monitor present communication error"("Register low" := "Modbus RTU buffer"."Monitor present communication error_L",   // "Concatenate two UInt into one UDInt"
                           "Register high" := "Modbus RTU buffer"."Monitor present communication error_H");
   #"Monitor communication error history 1"("Register low" := "Modbus RTU buffer"."Monitor communication error history 1_L",   // "Concatenate two UInt into one UDInt"
                           "Register high" := "Modbus RTU buffer"."Monitor communication error history 1_H");
   #"Monitor communication error history 2"("Register low" := "Modbus RTU buffer"."Monitor communication error history 2_L",   // "Concatenate two UInt into one UDInt"
                           "Register high" := "Modbus RTU buffer"."Monitor communication error history 2_H");
   #"Monitor communication error history 3"("Register low" := "Modbus RTU buffer"."Monitor communication error history 3_L",   // "Concatenate two UInt into one UDInt"
                           "Register high" := "Modbus RTU buffer"."Monitor communication error history 3_H");
   #"Monitor communication error history 4"("Register low" := "Modbus RTU buffer"."Monitor communication error history 4_L",   // "Concatenate two UInt into one UDInt"
                           "Register high" := "Modbus RTU buffer"."Monitor communication error history 4_H");
   #"Monitor communication error history 5"("Register low" := "Modbus RTU buffer"."Monitor communication error history 5_L",   // "Concatenate two UInt into one UDInt"
                           "Register high" := "Modbus RTU buffer"."Monitor communication error history 5_H");
   #"Monitor feedback position"("Register low" := "Modbus RTU buffer"."Monitor feedback position_L",   // "Concatenate two UInt into one UDInt"
                           "Register high" := "Modbus RTU buffer"."Monitor feedback position_H");
   #"Monitor feedback speed r/min"("Register low" := "Modbus RTU buffer"."Monitor feedback speed r/min_L",   // "Concatenate two UInt into one UDInt"
                           "Register high" := "Modbus RTU buffer"."Monitor feedback speed r/min_H");
   #"Monitor feedback speed Hz"("Register low" := "Modbus RTU buffer"."Monitor feedback speed Hz_L",   // "Concatenate two UInt into one UDInt"
                           "Register high" := "Modbus RTU buffer"."Monitor feedback speed Hz_H");
   #"Monitor direct I/O"("Register low" := "Modbus RTU buffer"."Monitor direct I/O_L",   // "Concatenate two UInt into one UDInt"
                         "Register high" := "Modbus RTU buffer"."Monitor direct I/O_H");
   #"Monitor torque"("Register low" := "Modbus RTU buffer"."Monitor torque_L",   // "Concatenate two UInt into one UDInt"
                     "Register high" := "Modbus RTU buffer"."Monitor torque_H");
   #"Monitor cumulative load"("Register low" := "Modbus RTU buffer"."Monitor cumulative load_L",   // "Concatenate two UInt into one UDInt"
                           "Register high" := "Modbus RTU buffer"."Monitor cumulative load_H");
   #"Monitor driver temperature"("Register low" := "Modbus RTU buffer"."Monitor driver temperature_L",   // "Concatenate two UInt into one UDInt"
                           "Register high" := "Modbus RTU buffer"."Monitor driver temperature_H");
   #"Monitor motor temperature"("Register low" := "Modbus RTU buffer"."Monitor motor temperature_L",   // "Concatenate two UInt into one UDInt"
                           "Register high" := "Modbus RTU buffer"."Monitor motor temperature_H");
   #"Monitor inverter voltage"("Register low" := "Modbus RTU buffer"."Monitor inverter voltage_L",   // "Concatenate two UInt into one UDInt"
                           "Register high" := "Modbus RTU buffer"."Monitor inverter voltage_H");
   #"Monitor power supply voltage"("Register low" := "Modbus RTU buffer"."Monitor power supply voltage_L",   // "Concatenate two UInt into one UDInt"
                           "Register high" := "Modbus RTU buffer"."Monitor power supply voltage_H");
   #"Monitor DIP SW"("Register low" := "Modbus RTU buffer"."Monitor DIP SW_L",   // "Concatenate two UInt into one UDInt"
                     "Register high" := "Modbus RTU buffer"."Monitor DIP SW_H");
   #"Monitor ROT SW0"("Register low" := "Modbus RTU buffer"."Monitor ROT SW0_L",   // "Concatenate two UInt into one UDInt"
                      "Register high" := "Modbus RTU buffer"."Monitor ROT SW0_H");
   #"Monitor ROT SW1"("Register low" := "Modbus RTU buffer"."Monitor ROT SW1_L",   // "Concatenate two UInt into one UDInt"
                      "Register high" := "Modbus RTU buffer"."Monitor ROT SW1_H");
END_REGION
END_FUNCTION_BLOCK
